// TIA Portal V17 export
// export: Created 2026-04-13T11:12:44.1316858Z, ExportSetting WithDefaults, DisplayName Totally Integrated Automation Portal, DisplayVersion V17 Update 4, DisplayName TIA Portal Openness, DisplayVersion V17 Update 4, DisplayName TIA Portal Version Control Interface, DisplayVersion V17, DisplayName SINAMICS Startdrive Advanced, DisplayVersion V17, DisplayName SINAMICS Startdrive G130, G150, S120, S150, SINAMICS MV, S210, DisplayVersion V17, DisplayName SINAMICS Startdrive G110M, G120, G120C, G120D, G120P, G115D, DisplayVersion V17, DisplayName STEP 7 Professional, DisplayVersion V17 Update 4, DisplayName STEP 7 Safety, DisplayVersion V17, DisplayName WinCC Professional, DisplayVersion V17 Update 4
FUNCTION_BLOCK "11-模拟量输出"   // FB55, SCL
{ S7_Optimized_Access := 'TRUE' }
VERSION : 0.1
// stored: AutoNumber true, IsIECCheckEnabled false, IsRetainMemResEnabled false, MemoryReserve 100, SetENOAutomatically false, UDAEnableTagReadback false
   VAR_INPUT
      HMI上限 : Real;
      HMI下限 : Real;
      PLC上限 : Int;
      PLC下限 : Int;
   END_VAR
   VAR_IN_OUT
      PLC调控 : Int;
      HMI设定 : Real;
   END_VAR
   VAR
      DBD1 : Real;
   END_VAR
BEGIN
   #DBD1 := NORM_X_REAL(MIN := #HMI下限, VALUE := #HMI设定, MAX := #HMI上限);
   #PLC调控 := SCALE_X_INT(MIN := #PLC下限, VALUE := #DBD1, MAX := #PLC上限);
END_FUNCTION_BLOCK
